Staubli VAL3: coord2Cell.pgx

program coord2Cell(num col_, num row_, string& x_sCellNumber[])
  local string strRow
  local string strCol
begin
  // transform row and column number to cell address string of camera
  // f.i. row = 2, col = 3 returns "C002"
  strRow=toString("0.0",row_)
  if row_<10
    strRow="0"+strRow
  endIf
  if row_<100
    strRow="0"+strRow
  endIf
  strCol=chr(col_+96)
  //
  x_sCellNumber=strCol+strRow
end
